// TIA Portal V20 export
TYPE "typeCmControlNodeCommand"
// stored: Namespace Unit1.Em8
   STRUCT
      thicknessAxisZ : "LER_typeAxisCommand";
      hipotThicknessServoPress { S7_SetPoint := 'True'} : "LER_typeServoPressCommand";
      hipotThicknessStageLiftFront { S7_SetPoint := 'True'} : "LER_typeTwoWayActCommand";
      hipotThicknessStageLiftRear { S7_SetPoint := 'True'} : "LER_typeTwoWayActCommand";
      hipotTabContactor { S7_SetPoint := 'True'} : "LER_typeTwoWayActCommand";
      hipotTabContactorLeft { S7_SetPoint := 'True'} : "LER_typeTwoWayActCommand";
      hipotTabContactorRight { S7_SetPoint := 'True'} : "LER_typeTwoWayActCommand";
      hipotThicknessStageLiftAll { S7_SetPoint := 'True'} : "LER_typeTwoWayActCommand";
   END_STRUCT;
END_TYPE
